  /// Server Invalid parameter value - TargetFrameNo outside of the allowed range 0..254 or does not exist on the RC
  /// Command "CalculateCartesianPosition"
  ERR_INVALID_PARAM_TARGET_FRAMENO_OUT_OF_RANGE := 16#8D72,

  /// Server Invalid parameter value - ToolNo outside of the allowed range 0..254 or does not exist on the RC
  /// Command "CalculateCartesianPosition"
  ERR_INVALID_PARAM_ERR_TOOLNO_INVALID := 16#8D73,

  /// Server Invalid parameter value - ParameterID does not exist on the RC
  /// Commands: "ReadSystemVariable", "WriteSystemVariable"
  ERR_INVALID_PARAM_PARAMETER_ID_INVALID := 16#8D74,

  /// Server Invalid parameter value - SubParameterID does not exist on the RC for the supplied ParameterID
  /// Commands: "ReadSystemVariable", "WriteSystemVariable"
  ERR_INVALID_PARAM_SUB_PARAMETER_ID_INVALID := 16#8D75,

  /// Server Invalid parameter value - SubParameterID must be 0 for a parameter without subparameters
  /// Commands: "ReadSystemVariable", "WriteSystemVariable"
  ERR_INVALID_PARAM_SUB_PARAMETER_MUST_BE_ZERO := 16#8D76,

  /// Server Invalid parameter value - SubParameterID must not be 0 for a parameter with subparameters
  /// Commands: "ReadSystemVariable", "WriteSystemVariable"
  ERR_INVALID_PARAM_SUB_PARAMETER_MUST_NOT_BE_ZERO := 16#8D77,

  /// Server Invalid parameter value - DataType outside of the allowed range 1..13
  /// Command "WriteSystemVariable"
  ERR_INVALID_PARAM_DATA_TYPE_OUT_OF_RANGE := 16#8D78,

  /// Server Invalid parameter value - DataType does not match the data type of the parameter
  /// Command "WriteSystemVariable"
  ERR_INVALID_PARAM_DATA_TYPE_MISMATCH := 16#8D79,

  /// Server Invalid parameter value - Data_0 contains invalid data for the target parameter
  /// Command "WriteSystemVariable"
  ERR_INVALID_PARAM_DATA_0_INVALID := 16#8D80,

  /// Server Invalid parameter value - Data_1 contains invalid data for the target parameter
  /// Command "WriteSystemVariable"
  ERR_INVALID_PARAM_DATA_1_INVALID := 16#8D81,

  /// Server Invalid parameter value - Data_2 contains invalid data for the target parameter
  /// Command "WriteSystemVariable"
  ERR_INVALID_PARAM_DATA_2_INVALID := 16#8D82,

  /// Server Invalid parameter value - Data_3 contains invalid data for the target parameter
  /// Command "WriteSystemVariable"
  ERR_INVALID_PARAM_DATA_3_INVALID := 16#8D83,

  /// Server Invalid parameter value - Data_4 contains invalid data for the target parameter
  /// Command "WriteSystemVariable"
  ERR_INVALID_PARAM_DATA_4_INVALID := 16#8D84,

  /// Server Invalid parameter value - Data_5 contains invalid data for the target parameter
  /// Command "WriteSystemVariable"
  ERR_INVALID_PARAM_DATA_5_INVALID := 16#8D85,

  /// Server Invalid parameter value - Data_6 contains invalid data for the target parameter
  /// Command "WriteSystemVariable"
  ERR_INVALID_PARAM_DATA_6_INVALID := 16#8D86,

  /// Server Invalid parameter value - Data_7 contains invalid data for the target parameter
  /// Command "WriteSystemVariable"
  ERR_INVALID_PARAM_DATA_7_INVALID := 16#8D87,

  /// Server Invalid parameter value - ReferenceFrame outside of the allowed range 0..254 or does not exist on the RC
  /// Command "CalculateFrame"
  ERR_INVALID_PARAM_REFERENCE_FRAME_OUT_OF_RANGE := 16#8D88,

  /// Server Optional parameter value not supported - DecelerationRate
  /// Commands using the parameter "DecelerationRate"
  ERR_OPTIONAL_PARAM_DECELERATION_RATE_NOT_SUPPORTED := 16#8E03,

  /// Server Optional parameter value not supported - JerkRate
  /// Commands using the parameter "JerkRate"
  ERR_OPTIONAL_PARAM_JERK_RATE_NOT_SUPPORTED := 16#8E04,

  /// Server Optional parameter value not supported - BlendingMode
  /// Commands using the parameter "BlendingMode"
  ERR_OPTIONAL_PARAM_BLENDING_MODE_NOT_SUPPORTED := 16#8E05,

  /// Server Optional parameter value not supported - Time
  /// Commands using the parameter "Time"
  ERR_OPTIONAL_PARAM_TIME_NOT_SUPPORTED := 16#8E06,

  /// Server Optional parameter value not supported - Position
  /// Commands using the parameter "Position"
  ERR_OPTIONAL_PARAM_POSITION_NOT_SUPPORTED := 16#8E07,

  /// Server Optional parameter value not supported - OriMode
  /// Commands using the parameter "OriMode"
  ERR_OPTIONAL_PARAM_ORI_MODE_NOT_SUPPORTED := 16#8E08,

  /// Server Optional parameter value not supported - ConfigMode
  /// Commands using the parameter "ConfigMode"
  ERR_OPTIONAL_PARAM_CONFIG_MODE_NOT_SUPPORTED := 16#8E09,

  /// Server Optional parameter value not supported - TurnMode
  /// Commands using the parameter "TurnMode"
  ERR_OPTIONAL_PARAM_TURN_MODE_NOT_SUPPORTED := 16#8E10,

  /// Server Optional parameter value not supported - TrajectoryMode
  /// Command "ReturnToPrimary"
  ERR_OPTIONAL_PARAM_TRAJECTORY_MODE_NOT_SUPPORTED := 16#8E11,

  /// Server Optional parameter value not supported - OperationMode
  /// Command "SetOperationMode"
  ERR_OPTIONAL_PARAM_OPERATION_MODE_NOT_SUPPORTED := 16#8E12,

  /// Server Optional parameter value not supported - IncrementalRotation
  /// Command "GroupJog"
  ERR_OPTIONAL_PARAM_INC_ROTATION_NOT_SUPPORTED := 16#8E13,

  /// Server Optional parameter value not supported - IncrementalTranslation
  /// Command "GroupJog"
  ERR_OPTIONAL_PARAM_INC_TRANSLATION_NOT_SUPPORTED := 16#8E14,

  /// Server Optional parameter value not supported - StepMode Exact Stop
  /// Command "EnableRobot"
  ERR_OPTIONAL_PARAM_STEP_MODE_EXACT_STOP_NOT_SUPPORTED := 16#8E16,

  /// Server Optional parameter value not supported - StepMode Blending
  /// Command "EnableRobot"
  ERR_OPTIONAL_PARAM_STEP_MODE_BLENDING_NOT_SUPPORTED := 16#8E17,

  /// Server Optional parameter value not supported - ModifiedConvention
  /// Command "ReadDHParameter"
  ERR_OPTIONAL_PARAM_MODIFIED_CONVENTION_NOT_SUPPORTED := 16#8E20,

  /// Server Optional parameter value not supported - WaitAtBlendingPoint
  /// Command "ExchangeConfig"
  ERR_OPTIONAL_PARAM_WAIT_AT_BLENDING_POINT_NOT_SUPPORTED := 16#8E21,

  /// Server Optional parameter not supported - Angle
  /// Commands: "MoveCircularAbsolute", "MoveCircularRelative", "MoveCircularCam"
  ERR_OPTIONAL_PARAM_ANGLE_NOT_SUPPORTED := 16#8E23,

  /// Server Optional parameter not supported - PathChoice
  /// Commands: "MoveCircularAbsolute", "MoveCircularRelative", "MoveCircularCam"
  ERR_OPTIONAL_PARAM_PATH_CHOICE_NOT_SUPPORTED := 16#8E24,

  /// Server Optional parameter not supported - Tolerance
  /// Commands: "MoveCircularAbsolute", "MoveCircularRelative", "MoveCircularCam"
  ERR_OPTIONAL_PARAM_TOLERANCE_NOT_SUPPORTED := 16#8E25,

  /// Server Optional parameter not supported - TransformationParameter_2
  /// Command "ShiftPosition"
  ERR_OPTIONAL_PARAM_TRANSFORMATION_PARAM2_NOT_SUPPORTED := 16#8E26,

  /// Server Optional parameter not supported - RotationAngle
  /// Command "ShiftPosition"
  ERR_OPTIONAL_PARAM_ROTATION_ANGLE_NOT_SUPPORTED := 16#8E27,

  /// Server Optional parameter value not supported - Mode
  /// Commands: "CalculateTool", "CalculateFrame"
  ERR_OPTIONAL_PARAM_VALUE_NOT_SUPPORTED := 16#8E28,

  /// Server Optional parameter not supported - ExternalTCP
  /// Commands: "CalculateTool", "CalculateFrame"
  ERR_OPTIONAL_PARAM_EXTERNAL_TCP_NOT_SUPPORTED := 16#8E29,

  /// Server Optional parameter not supported - RelativePosition
  /// Commands using the parameter "RelativePosition"
  ERR_OPTIONAL_PARAM_RELATIVE_POS_NOT_SUPPORTED := 16#8E30,

  /// Server Specified Emitter ID must not be 0
  /// Commands using the parameter "EmitterID"
  ERR_EMITTER_ID_MUST_NOT_BE_ZERO := 16#8F04,

  /// Server Invalid parameter value - Execution mode
  /// All Commands
  ERR_INVALID_PARAM_EXECUTION_MODE := 16#8F10,

  /// Server Command not implemented
  /// All Commands
  ERR_CMD_NOT_IMPLEMENTED := 16#8F11,

  /// Server Only one instance of this command is allowed
  /// Commands: "EnableRobot", "GroupJog", "ReturnToPrimary", "ExchangeConfig"
  ERR_CMD_ONLY_ONE_INSTANCE_ALLOWED := 16#8F12,

  /// Server Command requires an active interrupt or idle state to be executed
  /// Commands: "GroupJog", "ReturnToPrimary"
  ERR_CMD_REQUIRES_INTERRUPT_OR_IDLE_STATE := 16#8F13,

  /// Server Command cannot be executed during active interrupt
  /// Command "ReturnToPrimary"
  ERR_CMD_NOT_ALLOWED_DURING_ACTIVE_INTERRUPT := 16#8F14,

  /// Server Secondary sequence is blocked by command (e.g. GroupJog, ReturnToPrimary). No other commands may be buffered in secondary sequence
  /// All commands processed in secondary sequence
  ERR_SECONDARY_SEQUENCE_BLOCKED_BY_CMD := 16#8F15,

  /// Server The secondary sequence is not active. Commands may only be buffered in this sequence if it is active
  /// Commands using the parameter "SequenceFlag"
  ERR_SECONDARY_SEQUENCE_NOT_ACTIVE := 16#8F16,

  /// Server Secondary sequence is not empty. The command requires the secondary sequence to be empty
  /// Commands: "GroupJog", "ReturnToPrimary"
  ERR_SECONDARY_SEQUENCE_NOT_EMPTY := 16#8F17,

  /// Server Transaction not possible in the state machine
  /// All commands
  ERR_TRANSACTION_NOT_POSSIBLE_IN_STATE_MACHINE := 16#8F18,

  /// Server Cannot execute command because current operation mode is local.
  /// Commands that are not available in local modes
  ERR_CMD_NOT_POSSIBLE_BY_OP_MODE_LOCAL := 16#8F19,

  /// Server Command type out of range
  /// All commands
  ERR_CMD_TYPE_OUT_OF_RANGE := 16#8F20,

  /// Server Execution of this CMD is not possible while CallSubprogram is in progress in the sequence
  /// Commands: "SetSequence", "GroupJog"
  ERR_CMD_NOT_POSSIBLE_DURING_CALL_SUB_PROGRAM := 16#8F21,

  /// Server Operation not possible. See MessageLog for further information
  /// All commands
  ERR_OPERATION_NOT_POSSIBLE_SEE_LOG := 16#8F36,

  /// Server An RC internal error occurred during execution of this command. Check the message log for additional information
  /// All commands
  ERR_INTERNAL_ERROR_DURING_CMD := 16#8FFF,
  
  /// 7.2 Table "B" – RI ErrorIDs
  /// RI errors can occur on the PLC as well as on the RC. In the event of an RI error on the PLC, the
  /// corresponding ErrorID is written to the PLC message buffer independent of the function call
  /// "ReadMessages". In the event of an RI error on the RC, the ErrorID is transmitted via the function
  /// block "ReadMessages" and is also stored in PLC message buffer.
  /// In the PLC message buffer, they are dynamically arranged by the client to be displayed as follows:
  /// <Origin> <MessageType> <Description>
  /// More information about the general message handling mechanism can be found in 5.5.11
  /// Diagnostics.
  /// The following table gives an overview over the existing "ErrorIDs" reported via RI errors and the
  /// corresponding description.

  /// ------------------------------------------------------
  /// Client ErrorIDs
  /// ------------------------------------------------------

  /// Client Wrong Telegram State (Two Sequences not in both directions active)
  ERR_WRONG_TELEGRAM_STATE  := 16#8001,

  /// Client Acyclic area client to server too small
  ERR_ACYCLIC_AREA_TO_SMALL_PLC_TO_ROB  := 16#8002,

  /// Client Acyclic area server to client too small
  ERR_ACYCLIC_AREA_TO_SMALL_ROB_TO_PLC := 16#8003,

  /// Client Lifesign timeout
  ERR_LIFESIGN_TIMEOUT_0x8005 := 16#8004,

  /// Client Telegram sequence timeout
  ERR_TELEGRAM_SEQ_TIMEOUT_0x8005 := 16#8005,

  /// Client Assigned AxesGroup not valid
  ERR_AXESGROUP_INVALID := 16#8007,

  /// Client Assigned periphery not valid
  ERR_PERIPHERY_INVALID := 16#8008,

  /// Client Invalid state of the robot (more than 1 CMD active)
  ERR_INVALID_ROBOT_STATE := 16#8009,

  /// Client Telegram Number changed after initialization. Reinitialize by disabling and enabling the RobotTask.
  ERR_TELEGRAM_NUMBER_CHANGED_AFTER_INIT  := 16#8013,
    
  /// Client Telegram control does not match the telegram state
  ERR_TELEGRAM_CONTROL_MISMATCH_TELEGRAM_STATE_0x80A1 := 16#80A1,

  /// Client Initialization lost for unknown reason. See message log after reinitializing
  ERR_INIT_LOST_UNKNOWN_0x80A2  := 16#80A2,

  /// Client Telegram length does not match the length provided in the communication interface, or the communication interface is too small.
  ERR_TELEGRAM_LENGTH_MISMATCH_0x80A3  := 16#80A3,

  /// Client Incompatible major SRCI version
  ERR_SRCI_MAJOR_VERSION_INCOMPATIBLE_0x80A4  := 16#80A4,

  /// Client Lifesign timeout
  ERR_LIFESIGN_TIMEOUT_0x80A5 := 16#80A5,

  /// Client The selected optional cyclic data does not fit in the given telegram size
  ERR_CYCLIC_DATA_TOO_LARGE_0x80A6  := 16#80A6,

  /// Client The robot interface was reset after being initialized
  ERR_INTERFACE_WAS_RESET_AFTER_INIT_0x80A7  := 16#80A7,

  /// Client Telegram sequence timeout
  ERR_TELEGRAM_SEQ_TIMEOUT_0x80A8_0x80A8  := 16#80A8,

  /// Client The telegram number changed after initialization
  ERR_TELEGRAM_NO_CHANGED_AFTER_INIT_0x80A9 := 16#80A9,

  /// Client Error: Invalid AxesGroupID
  ERR_AXESGROUP_ID_INVALID_0x80AA  := 16#80AA,

  /// Client Telegram number is invalid. E.g. TwoSequences is only activated in one direction
  ERR_TELEGRAM_NUMBER_INVALID_0x80AB  := 16#80AB,

  /// Client Telegram Number is not supported
  ERR_TELEGRAM_NUMBER_NOT_SUPPORTED_0x80AC := 16#80AC,

  /// Server The ACR is full. RA is disabled
  ERR_ACR_REGISER_IS_FULL  := 16#8A01,

  /// Server The execution of a mandatory command has been stopped. Exchange config must run for the system to run
  ERR_MANDATORY_CMD_STOPPED  := 16#8A02,

  /// Server Inconsistent data received. Make sure the complete telegram data is sent to RC in one frame.
  ERR_INCONSISTENT_DATA_RECEIVED  := 16#8A03,

  /// Client Connection to the communication partner was lost
  ERR_CONNECTION_LOST  := 16#8AAD,

  /// Client Fatal Error occurred. Reinitialization of Robot_Task is required
  ERR_FATAL_ERROR_REINIT_REQUIRED  := 16#9001,

  /// ------------------------------------------------------
  /// SERVER ErrorIDs
  /// ------------------------------------------------------
  
  /// Server Internal error
  ERR_INTERNAL_ERROR  := 16#9A01,

  /// Server Internal error in deserialize
  ERR_DESERIALIZE_ERROR  := 16#9A02,

  /// Server CMD ID out of range 1.ACR_Length
  ERR_CMD_ID_OUT_OF_RANGE  := 16#9A03,

  /// Server Invalid fragment length
  ERR_FRAGMENT_LENGTH_INVALID := 16#9A04,

  /// Server Command priority or type changed during runtime
  ERR_CMD_PRIORITY_CHANGED := 16#9A05,

  /// Server Tried to reset a non-empty ACR entry
  ERR_TRIED_TO_RESET_NONEMPTY_ACR_REGISTER := 16#9A06,

  /// Server Error: Invalid Sequence payload length (e.g., sequence payload length is specified 999 even if telegram length is only 100.)
  ERR_SEQUENCE_PAYLOAD_INVALID_LENGTH := 16#9A07,

  /// Server Invalid ActionByte
  ERR_ACTION_BYTE_INVALID := 16#9A08,

  /// Server Invalid Command payload length
  ERR_CMD_PAYLOAD_LENGTH_INVALID := 16#9A09,

  /// Server Error: Invalid Command payload pointer (e.g., Out of bounds)
  ERR_CMD_PAYLOAD_POINTER_INVALID := 16#9A10,

  /// Server Illegal Execution Mode change
  ERR_EXEC_MODE_CHANGE_ILLEGAL := 16#9A14

)WORD;
END_TYPE

// Library/Enumerations/Events/RobotLibraryInfoIdEnum
{attribute 'qualified_only'}
TYPE RobotLibraryInfoIdEnum :
(
  NO_INFO := 0,
  
  ////7.5 Table "E" – Command InfoIDs
  /// If an info event related to the execution of a function block occurs, the function block returns an
  /// InfoID to specify the event. The info events are stored in the PLC message buffer and are displayed
  /// on the function block outputs.
  /// In the PLC message buffer, they are dynamically arranged by the client to be displayed as follows:
  /// <Origin> <MessageType> <Command name> <Description>
  /// More information about the general message handling mechanism can be found in 5.5.11
  /// Diagnostics.
  /// The following table gives an overview over the existing InfoIDs reported by commands and the
  /// corresponding description.

  /// Server Collision detected
  /// Motion commands
  INFO_COLLISION_DETECTED := 16#6C01,

  /// Server Error occurred during motion. Check the message buffer for more information
  /// Motion commands
  INFO_MOTION_ERROR := 16#6C02,

  /// Server Target position not reachable
  /// Motion commands
  INFO_TARGET_POS_UNREACHABLE := 16#6C03,

  /// Server Software limits reached
  /// Motion commands
  INFO_SW_LIMITS_REACHED := 16#6C04,

  /// Server Abortion of this command was requested by a GroupStop
  /// All sequence related commands
  INFO_ABORT_BY_GROUP_STOP := 16#6C05,

  /// Server Abortion of this command was requested by another motion command
  /// All sequence related commands
  INFO_ABORT_BY_MOTION_CMD := 16#6C06,

  /// Server Reading the currently used software limits. Updated software limits are active after restart.
  /// Command "ReadRobotSWLimits"
  INFO_READ_SW_LIMITS := 16#6C07,

  /// Server No SubProgram was stopped because none was active
  /// Command "StopSubprogram"
  INFO_NO_ACTIVE_SUBPROGRAM := 16#6C09,

  /// Server A program for the supplied JobID is not running or does not exist.
  /// Command "StopSubprogram"
  INFO_JOBID_NOT_RUNNING := 16#6C11,

  /// Server A program for the supplied InstanceID is not running or does not exist.
  /// Command "StopSubprogram"
  INFO_INSTANCEID_NOT_RUNNING := 16#6C12,

  /// Server The robot is waiting at the blending zone.
  /// Motion commands
  INFO_WAITING_AT_BLEND_ZONE := 16#6C13,

  /// Server Jog motion was interrupted by GroupStop
  /// Command "GroupJog"
  INFO_JOG_INTERRUPTED_BY_GROUP_STOP := 16#6C14,

  /// Server Jog motion was interrupted by RA sequence state INTERRUPTED
  /// Command "GroupJog"
  INFO_JOG_INTERRUPTED_BY_RA_STATE := 16#6C15,

  /// Server Manual start is ignored when the sequence is empty
  /// Command "EnableRobot"
  INFO_MANUAL_START_IGNORED_DURING_EMPTY_SEQ := 16#6C19,

  /// Server Invalid parameter value - A value was given for index 0. Index 0 is not writeable. Remove the value or change the index.
  /// Commands: "WriteIntegers", "WriteReals", "WriteAnalogOutputs", "ReadDigitalInputs", "ReadDigitalOutputs", "ReadIntegers", "ReadReals"
  INFO_PARAM_INDEX_ZERO_NOT_WRITEABLE := 16#6D51,

  /// Server Invalid parameter value OutputBitmask - No bitmask was given for a non zero index. Set the index to zero, or set a valid bitmask.
  /// Command "WriteDigitalOutputs"
  INFO_PARAM_OUTPUT_BITMASK_INVALID_FOR_NON_ZERO_INDEX := 16#6D52,

  /// Server Invalid parameter value OutputBitmask - A bitmask was given for a zero index. Set the bitmask to zero, or set a non zero index.
  /// Command "WriteDigitalOutputs"
  INFO_PARAM_OUTPUT_BITMASK_INVALID_FOR_ZERO_INDEX := 16#6D53,

  /// Server Command interrupted due to RA sequence state INTERRUPTED
  /// All sequence related commands
  INFO_CMD_INTERRUPTED_BY_RA_STATE  := 16#6F01,

  /// Server Command interrupted due to RA power state NOT_ENABLED
  /// All sequence related commands
  INFO_CMD_INTERRUPTED_BY_RA_NOT_ENABLED  := 16#6F02,

  /// Server Command interrupted due to RA sequence state INTERRUPTED while single step mode is active
  /// All sequence related commands
  INFO_CMD_INTERRUPTED_BY_RA_SEQ_STATE_DURING_STEP_MODE  := 16#6F03,

  /// Server Internal code used to reset warnings
  /// All commands
  INFO_RESET_WARNINGS_BY_INTERNAL_CODE  := 16#FF,


  /// 7.6 Table "F" – RI InfoIDs
  /// RI info events can occur on the PLC as well as on the RC. In the event of an RI info on the PLC,
  /// the corresponding InfoID is written to the PLC message buffer independent of the function call
  /// "ReadMessages". In the event of an RI info on the RC, the InfoID is transmitted via the function
  /// block "ReadMessages" and is also stored in PLC message buffer.
  /// In the PLC message buffer, they are dynamically arranged by the client to be displayed as follows:
  /// <Origin> <MessageType> <Description>
  /// More information about the general message handling mechanism can be found in 5.5.11
  /// Diagnostics.
  /// The following table gives an overview over the existing InfoIDs reported via RI info events and the
  /// corresponding description.  

  /// Client Lifesign smaller than lower limit. It has been increased to 10ms.
  INFO_LIFESIGN_TIMEOUT_TO_SMALL_AND_SET_TO_10MS  := 16#6001,

  /// Client ReceiveExtendedCartesianPosition cannot be used without ReceiveCartesianPos. RecCarPos is automatically activated.
  INFO_RECV_EXT_CART_POS_NOT_USABLE_WITH_RECV_CART_POS := 16#6002,

  /// Client ReceiveExtendedJointPosition cannot be used without ReceiveJointPosition. RecJointPos is automatically activated.
  INFO_RECV_EXT_JOINT_POS_NOT_USABLE_WITH_RECV_JOINT_POS := 16#6003,

  /// Client Synchronization of tool data is disabled, and the data is different on the RC. Tool = "NUMBER" (Please Enter a valid SyncMode)
  INFO_SYNC_TOOL_DATA_DISABLED  := 16#6014,

  /// Client Change the Syncmode to Negative only works on Startup with PLC (TOOL)
  INFO_CHANGE_TOOL_SYNC_MODE_TO_NEGATIVE_ONLY_AT_PLC_START_ALLOWED := 16#6015,

  /// Client Synchronization of frame data is disabled, and the data is different on the RC. Frame = "NUMBER" (Please Enter a valid SyncMode)
  INFO_SYNC_FRAME_DATA_DISABLED := 16#6020,

  /// Client Change the Syncmode to Negative only works on Startup with PLC (FRAME)
  INFO_CHANGE_FRAME_SYNC_MODE_TO_NEGATIVE_ONLY_AT_PLC_START_ALLOWED := 16#6021,

  /// Client Synchronization of load data is disabled, and the data is different on the RC. Load = "NUMBER" (Please Enter a valid SyncMode)
  INFO_SYNC_LOAD_DATA_DISABLED := 16#6026,

  /// Client Change the Syncmode to Negative only works on Startup with PLC (LOAD)
  INFO_CHANGE_LOAD_SYNC_MODE_TO_NEGATIVE_ONLY_AT_PLC_START_ALLOWED := 16#6027,

  /// Client Synchronization of work area data is disabled, and the data is different on the RC. WorkArea = "NUMBER" (Please Enter a valid SyncMode)
  INFO_SYNC_WORK_AREA_DISABLED := 16#6032,

  /// Client Change the Syncmode to Negative only works on Startup with PLC (WORKAREA)
  INFO_CHANGE_WORK_AREA_SYNC_MODE_TO_NEGATIVE_ONLY_AT_PLC_START_ALLOWED := 16#6033,

  /// Client Synchronization of Software Limits data is disabled, and the data is different on the RC.
  INFO_SYNC_SWLIMIT_DISABLED := 16#6036,

  /// Client Change the Syncmode to Negative only works on Startup with PLC (SW LIMITS)
  INFO_CHANGE_SWLIMITS_SYNC_MODE_TO_NEGATIVE_ONLY_AT_PLC_START_ALLOWED := 16#6037,

  /// Client Synchronization of default dynamics data is disabled, and the data is different on the RC.
  INFO_SYNC_DEFAULT_DYNAMICS_DISABLED := 16#6040,

  /// Client Change the Syncmode to Negative only works on Startup with PLC (DEFAULT DYNAMICS)
  INFO_CHANGE_DEFAULT_DYNAMIVS_SYNC_MODE_TO_NEGATIVE_ONLY_AT_PLC_START_ALLOWED := 16#6041,

  /// Client Synchronization of reference dynamics data is disabled, and the data is different on the RC.
  INFO_SYNC_REFERENCE_DYNAMICS_DISABLED := 16#6044,

  /// Client Change the Syncmode to Negative only works on Startup with PLC (REFERENCE DYNAMICS)
  INFO_CHANGE_REFERENCE_DYNAMIVS_SYNC_MODE_TO_NEGATIVE_ONLY_AT_PLC_START_ALLOWED := 16#6045,

  /// Server RA disabled due to operation mode change
  INFO_RA_DISABLED_BY_OPMODE_CHANGE  := 16#6A01,

  /// Server Operation mode changed
  INFO_OPERATION_MODE_CHANGED  := 16#6A02,

  /// Server The server state has been reset on client request. Client restart may be a cause.
  INFO_SERVER_STATE_RESET_BY_CLIENT_REQUEST  := 16#6A03,

  /// Server The actual override has been decreased to not exceed a movement's monitoring velocity.
  INFO_OVERRIDE_DECREASED_TO_PREVENT_EXEEDING_MONITORING_VELOCITY  := 16#6A07,

  /// Server Excessive logging may degrade system performance.
  INFO_EXCESSIVE_LOGGING  := 16#6A13,

  /// Server The first motion is executed with reduced velocity.
  INFO_FIRST_MOTION_REDUCED_VELOCITY  := 16#6C08
)WORD;
END_TYPE

// Library/Enumerations/Events/RobotLibraryWarningIdEnum
{attribute 'qualified_only'}
TYPE RobotLibraryWarningIdEnum :
(
  NO_WARNING := 0,
 
  /// 7.3 Table "C" – Command WarningIDs
  /// If a warning related to the execution of a function block occurs, the function block returns a
  /// WarningID to specify the warning. The warnings are stored in the PLC message buffer and are
  /// displayed on the function block outputs.
  /// In the PLC message buffer, they are dynamically arranged by the client to be displayed as follows:
  /// <Origin> <MessageType> <Command name> <Description>
  /// More information about the general message handling mechanism can be found in 5.5.11
  /// Diagnostics.
  /// The following table gives an overview over the existing WarningIDs reported by commands and
  /// the corresponding description.

  /// Client HighPriority Input is ignored when a sequential ProcessingMode is selected
  /// Commands: "WriteDigitalOutputs", "WriteIntegers", "WriteReals", "WriteAnalogOutputs"
  WARN_HIGHPRIORITY_IGNORED_SEQ_MODE  := 16#7301,

  /// Client Optional Cyclic data was disabled by the user but is still enabled until reinitialization of RobotTask
  /// Command: "ReadActualPositionCyclic"
  WARN_CYCLIC_DATA_DISABLED_STILL_ACTIVE  := 16#7303,

  /// Client Number of free entries in the ACR is running out
  /// All commands
  WARN_ACR_FREE_ENTRIES_LOW  := 16#7605,

  /// Server The Frame is currently used in the sequence
  /// Command: "WriteFrameData"
  WARN_FRAME_USED_IN_SEQUENCE  := 16#7C03,

  /// Server The Tool is currently used in the sequence
  /// Command: "WriteToolData"
  WARN_TOOL_USED_IN_SEQUENCE  := 16#7C04,

  /// Server The Load is currently used in the sequence
  /// Command: "WriteLoadData"
  WARN_LOAD_USED_IN_SEQUENCE  := 16#7C06,

  /// Server The monitoring does not apply to motion CMDs which are already buffered.
  /// Command: "SetTriggerMotion"
  WARN_MONITORING_DOES_NOT_APPLY_TO_BUFFERED_CMDS  := 16#7C14,

  /// 7.4 Table "D" – RI WarningIDs
  /// RI warnings can occur on the PLC as well as on the RC. In the event of an RI warning on the PLC,
  /// the corresponding WarningID is written to the PLC message buffer independent of the function call
  /// "ReadMessages". In the event of an RI warning on the RC, the WarningID is transmitted via the
  /// function block "ReadMessages" and is also stored in PLC message buffer.
  /// In the PLC message buffer, they are dynamically arranged by the client to be displayed as follows:
  /// <Origin> <MessageType> <Description>
  /// More information about the general message handling mechanism can be found in 5.5.11
  /// Diagnostics.
  /// The following table gives an overview over the existing WarningIDs reported via RI warnings and
  /// the corresponding description.

  /// Client Acyclic range client to server very small
  WARN_ACYCLIC_RANGE_PLC_TO_ROB_VERY_SMALL  := 16#7001,

  /// Client Acyclic range server to client very small
  WARN_ACYCLIC_RANGE_ROB_TO_PLC_VERY_SMALL := 16#7002,

  /// Client Telegram number was changed during operation
  WARN_TELEGRAM_NO_CHANGED_DURING_OPERATION  := 16#7003,

  /// Client Save Tool locally failed. Index not available in user data.
  WARN_SAVE_TOOL_FAILED := 16#7005,

  /// Client Save Frame locally failed. Index not available in user data.
  WARN_SAVE_FRAME_FAILED  := 16#7006,

  /// Client Save Load locally failed. Index not available in user data.
  WARN_SAVE_LOAD_FAILED  := 16#7007,

  /// Client Save WorkArea locally failed. Index not available in user data.
  WARN_SAVE_WORKAREA_FAILED  := 16#7008,

  /// Client Array of tool data supplied to RobotTask does not start at 0.
  WARN_TOOL_DATA_ARRAY_NOT_START_AT_ZERO  := 16#7009,

  /// Client Array of tool data supplied to RobotTask must be longer than the number of tools on the RC.
  WARN_TOOL_DATA_ARRAY_TOO_SHORT := 16#7010,

  /// Client Tool data sync mode is invalid.
  WARN_TOOL_DATA_SYNC_MODE_INVALID  := 16#7011,

  /// Client Error Sync with Tool "NUMBER" (Please Enter a valid SyncMode)
  WARN_TOOL_NUMBER_SYNC_ERROR  := 16#7012,

  /// Client Error Sync Data changed in both Sides with Tool "NUMBER" (Please Enter a valid SyncMode)
  WARN_TOOL_SYNC_BOTH_SIDES_CHANGED  := 16#7013,

  /// Client Array of frame data supplied to RobotTask does not start at 0.
  WARN_FRAME_DATA_ARRAY_NOT_START_AT_ZERO := 16#7015,

  /// Client Array of frame data supplied to RobotTask must be longer than the number of frames on the RC.
  WARN_FRAME_DATA_ARRAY_TOO_SHORT := 16#7016,

  /// Client Frame data sync mode is invalid.
  WARN_FRAME_DATA_SYNC_MODE_INVALID := 16#7017,

  /// Client Error Sync with Frame "NUMBER" (Please Enter a valid SyncMode)
  WARN_FRAME_NUMBER_SYNC_ERROR := 16#7018,

  /// Client Error Sync Data changed in both Sides with Frame "NUMBER" (Please Enter a valid SyncMode)
  WARN_FRAME_SYNC_BOTH_SIDES_CHANGED := 16#7019,

  /// Client Array of load data supplied to RobotTask does not start at 0.
  WARN_LOAD_DATA_ARRAY_NOT_START_AT_ZERO := 16#7021,

  /// Client Array of load data supplied to RobotTask must be longer than the number of tools on the RC.
  WARN_LOAD_DATA_ARRAY_TOO_SHORT := 16#7022,

  /// Client Load data sync mode is invalid.
  WARN_LOAD_DATA_SYNC_MODE_INVALID := 16#7023,

  /// Client Error Sync with Load "NUMBER" (Please Enter a valid SyncMode)
  WARN_LOAD_NUMBER_SYNC_ERROR := 16#7024,

  /// Client Error Sync Data changed in both Sides with Load "NUMBER" (Please Enter a valid SyncMode)
  WARN_LOAD_SYNC_BOTH_SIDES_CHANGED := 16#7025,

  /// Client Array of workarea data supplied to RobotTask does not start at 0.
  WARN_WORK_AREA_ARRAY_NOT_START_AT_ZERO := 16#7027,

  /// Client Array of workarea data supplied to RobotTask must be longer than the number of tools on the RC.
  WARN_WORK_AREA_ARRAY_TOO_SHORT := 16#7028,

  /// Client Workarea data sync mode is invalid.
  WARN_WORK_AREA_SYNC_MODE_INVALID := 16#7029,

  /// Client Error Sync with WorkArea "NUMBER" (Please Enter a valid SyncMode)
  WARN_WORK_AREA_NUMBER_SYNC_ERROR:= 16#7030,

  /// Client Error Sync Data changed in both Sides with WorkArea "NUMBER" (Please Enter a valid SyncMode)
  WARN_WORK_AREA_SYNC_BOTH_SIDES_CHANGED := 16#7031,

  /// Client Software limits data sync mode is invalid.
  WARN_SW_LIMITS_SYNC_MODE_INVALID := 16#7033,

  /// Client Error Sync with Software Limits (Please Enter a valid SyncMode)
  WARN_SW_LIMITS_SYNC_ERROR := 16#7034,

  /// Client Error Sync Data changed in both Sides with Software Limits (Please Enter a valid SyncMode)
  WARN_SW_LIMITS_SYNC_BOTH_SIDES_CHANGED := 16#7035,

  /// Client Default dynamics data sync mode is invalid.
  WARN_DEFAULT_DYNAMICS_SYNC_MODE_INVALID := 16#7037,

  /// Client Error Sync with Default Dynamics (Please Enter a valid SyncMode)
  WARN_DEFAULT_DYNAMICS_SYNC_ERROR := 16#7038,

  /// Client Error Sync Data changed in both Sides with Default Dynamics (Please Enter a valid SyncMode)
  WARN_DEFAULT_DYNAMICS_SYNC_BOTH_SIDES_CHANGED := 16#7039,

  /// Client Reference dynamics data sync mode is invalid.
  WARN_REFERENCE_DYNAMICS_SYNC_MODE_INVALID := 16#7041,

  /// Client Error Sync with Reference Dynamics (Please Enter a valid SyncMode)
  WARN_REFERENCE_DYNAMICS_SYNC_ERROR:= 16#7042,

  /// Client Error Sync Data changed in both Sides with Reference Dynamics (Please Enter a valid SyncMode)
  WARN_REFERENCE_DYNAMICS_SYNC_BOTH_SIDES_CHANGED := 16#7043,

  /// Client Synchronization of tool is not possible due to error in the read or write tool cmd. See dedicated message log entry for more information.
  WARN_TOOL_SYNC_FAILED_BY_ERROR_OF_READ_OR_WRITE_CMD  := 16#7044,

  /// Client Synchronization of frame is not possible due to error in the read or write frame cmd. See dedicated message log entry for more information.
  WARN_FRAME_SYNC_FAILED_BY_ERROR_OF_READ_OR_WRITE_CMD := 16#7045,

  /// Client Synchronization of load is not possible due to error in the read or write load cmd. See dedicated message log entry for more information.
  WARN_LOAD_SYNC_FAILED_BY_ERROR_OF_READ_OR_WRITE_CMD := 16#7046,

  /// Client Synchronization of swLimits is not possible due to error in the read or write swLimits cmd. See dedicated message log entry for more information.
  WARN_SW_LIMITS_SYNC_FAILED_BY_ERROR_OF_READ_OR_WRITE_CMD := 16#7047,

  /// Client Synchronization of referenceDynamics is not possible due to error in the read or write referenceDynamics cmd. See dedicated message log entry for more information.
  WARN_REFERENCE_DYNAMICS_SYNC_FAILED_BY_ERROR_OF_READ_OR_WRITE_CMD := 16#7048,

  /// Client Synchronization of defaultDynamics is not possible due to error in the read or write defaultDynamics cmd. See dedicated message log entry for more information.
  WARN_DEFAULT_DYNAMICS_SYNC_FAILED_BY_ERROR_OF_READ_OR_WRITE_CMD := 16#7049,

  /// Client Using the legacy SRCI version encoding. It will not be compatible with the newest RC interpreter versions.
  WARN_LEGACY_SRCI_ENCODING  := 16#7050,

  /// Server The ACR is almost full. Filling it completely disables the robot. Make sure to limit the number of commands in the system.
  WARN_ACR_ALMOST_FULL  := 16#7A01
)WORD;
END_TYPE

// Library/Enumerations/Flag/SequenceFlag
{attribute 'qualified_only'}
// ------------------------------------------------------------------------- 
//  SRCI Robot Library                                                
// ------------------------------------------------------------------------- 
//                                                                           
//  Object:      SequenceFlag                                       
//  Author:      Thorsten Brach                                                
//  Date:        2024-06-01
//
//  Description:                                              
//   
//                                                                           
//  Copyright: 
//    (C) 2024 Thorsten Brach. All rights reserved                                                                                                                                            
//             Licensed under the LGPL-3.0 license.
//                                                                           
//  Disclaimer:                                                                           
//    This project is provided without any guarantee and can be used for   
//    private and commercial purposes. Any use is at the user’s 
//    own risk and responsibility.
//
// -------------------------------------------------------------------------
TYPE SequenceFlag :
(
  /// • Refers to ProcessingModes 2 to 5 and 9 (2 = Parallel, 3 = Continuous, 4 = not available, 5 = Trigger Multiple, 9 = Deactivate )
  /// • Command is not handled by any sequence
  /// • For more information on ProcessingModes refer to chapter 5.6.4.5
  NO_SEQUENCE := 0,
  /// • Command will be handled by primary sequence
  PRIMARY_SEQUENCE := 1,
  /// • Command will be handled by secondary sequence
  SECONDARY_SEQUENCE := 2
)USINT;
END_TYPE

// Library/Enumerations/Level/LogLevel
{attribute 'qualified_only'}
// ------------------------------------------------------------------------- 
//  SRCI Robot Library                                                
// ------------------------------------------------------------------------- 
//                                                                           
//  Object:      LogLevel                                       
//  Author:      Thorsten Brach                                                
//  Date:        2024-06-01
//
//  Description:                                              
//   
//                                                                           
//  Copyright: 
//    (C) 2024 Thorsten Brach. All rights reserved                                                                                                                                            
//             Licensed under the LGPL-3.0 license.
//                                                                           
//  Disclaimer:                                                                           
//    This project is provided without any guarantee and can be used for   
//    private and commercial purposes. Any use is at the user’s 
//    own risk and responsibility.
//
// -------------------------------------------------------------------------
TYPE LogLevel : Severity; END_TYPE

// Library/Enumerations/Level/LogLevelEnum
TYPE LogLevelEnum : LogLevel; END_TYPE

// Library/Enumerations/Level/MessageLevel
{attribute 'qualified_only'}
// ------------------------------------------------------------------------- 
//  SRCI Robot Library                                                
// ------------------------------------------------------------------------- 
//                                                                           
//  Object:      MessageLevel                                       
//  Author:      Thorsten Brach                                                
//  Date:        2024-06-01
//
//  Description:                                              
//   
//                                                                           
//  Copyright: 
//    (C) 2024 Thorsten Brach. All rights reserved                                                                                                                                            
//             Licensed under the LGPL-3.0 license.
//                                                                           
//  Disclaimer:                                                                           
//    This project is provided without any guarantee and can be used for   
//    private and commercial purposes. Any use is at the user’s 
//    own risk and responsibility.
//
// -------------------------------------------------------------------------
TYPE MessageLevel :
(
  /// Debugging messages, Informative messages, Warning messages, Error messages, Fatal error messages
  DEBUG := 4,
  /// Informative messages, Warning messages, Error messages, Fatal error messages 
  INFO := 5, 
  /// Warning messages, Error messages, Fatal error messages
  WARNING := 20,
  /// Error messages, Fatal error messages 
  ERROR := 28 
)USINT;
END_TYPE

// Library/Enumerations/Level/PriorityLevel
{attribute 'qualified_only'}
// ------------------------------------------------------------------------- 
//  SRCI Robot Library                                                
// ------------------------------------------------------------------------- 
//                                                                           
//  Object:      PriorityLevel                                       
//  Author:      Thorsten Brach                                                
//  Date:        2024-06-01
//
//  Description:                                              
//   
//                                                                           
//  Copyright: 
//    (C) 2024 Thorsten Brach. All rights reserved                                                                                                                                            
//             Licensed under the LGPL-3.0 license.
//                                                                           
//  Disclaimer:                                                                           
//    This project is provided without any guarantee and can be used for   
//    private and commercial purposes. Any use is at the user’s 
//    own risk and responsibility.
//
// -------------------------------------------------------------------------
TYPE PriorityLevel :
(
  /// priority level is very high 
  VERY_HIGH := 1,
  /// priority level is high 
  HIGH := 2,
  /// priority level is normal 
  NORMAL := 3,
  /// priority level is low 
  LOW := 4  
)BYTE;
END_TYPE

// Library/Enumerations/Miscellaneous/CircPlane
{attribute 'qualified_only'}
{attribute 'strict'}
// ------------------------------------------------------------------------- 
//  SRCI Robot Library                                                
// ------------------------------------------------------------------------- 
//                                                                           
//  Object:      CircPlane                                       
//  Author:      Thorsten Brach                                                
//  Date:        2024-06-01
//
//  Description:                                              
//   
//                                                                           
//  Copyright: 
//    (C) 2024 Thorsten Brach. All rights reserved                                                                                                                                            
//             Licensed under the LGPL-3.0 license.
//                                                                           
//  Disclaimer:                                                                           
//    This project is provided without any guarantee and can be used for   
//    private and commercial purposes. Any use is at the user’s 
//    own risk and responsibility.
//
// -------------------------------------------------------------------------
TYPE CircPlane :
(
  /// x-z-plane
  XZ_PLANE := 0,
  /// y-z-plane
  YZ_PLANE := 1,
  /// x-y-plane
  XY_PLANE := 2
)SINT;
END_TYPE

// Library/Enumerations/Miscellaneous/ControlHalfByte
{attribute 'qualified_only'}
// ------------------------------------------------------------------------- 
//  SRCI Robot Library                                                
// ------------------------------------------------------------------------- 
//                                                                           
//  Object:      ControlHalfByte                                       
//  Author:      Thorsten Brach                                                
//  Date:        2024-06-01
//
//  Description:                                              
//   
//                                                                           
//  Copyright: 
//    (C) 2024 Thorsten Brach. All rights reserved                                                                                                                                            
//             Licensed under the LGPL-3.0 license.
//                                                                           
//  Disclaimer:                                                                           
//    This project is provided without any guarantee and can be used for   
//    private and commercial purposes. Any use is at the user’s 
//    own risk and responsibility.
//
// -------------------------------------------------------------------------
TYPE ControlHalfByte :
(
  /// Default value, no control active
  NONE := 0,
  /// Initialization is requested by the client
  INITIALIZE := 1,
  /// Resume of operation is requested by the client
  RESUME := 2,
  /// Resetting of the RC is requested by the client. The RC must stop the motion, and clear all state.
  RESET := 3,
  /// Acknowledgement of a telegram state error
  ACK_ERROR := 4,
  /// Signaling that a client error occurred. The Server must respond by setting its RI state to NOT_INITIALIZED
  CLIENT_ERROR := 5
)BYTE;
END_TYPE

// Library/Enumerations/Miscellaneous/ErrorReaction
{attribute 'qualified_only'}
// ------------------------------------------------------------------------- 
//  SRCI Robot Library                                                
// ------------------------------------------------------------------------- 
//                                                                           
//  Object:      ErrorReaction                                       
//  Author:      Thorsten Brach                                                
//  Date:        2024-06-01
//
//  Description:                                              
//   
//                                                                           
//  Copyright: 
//    (C) 2024 Thorsten Brach. All rights reserved                                                                                                                                            
//             Licensed under the LGPL-3.0 license.
//                                                                           
//  Disclaimer:                                                                           
//    This project is provided without any guarantee and can be used for   
//    private and commercial purposes. Any use is at the user’s 
//    own risk and responsibility.
//
// -------------------------------------------------------------------------
TYPE ErrorReaction :
(
  /// Abort and move Abort active move command and delete commands buffered in sequence Move robot by specified ErrorVector
  ABORT_AND_MOVE := 0,
  /// 1: Abort
  /// Abort active move command and delete commands buffered in sequence
  /// No additional movements
  ABORT := 1,  
  /// 2: No reaction
  /// Error event is ignored by active move command
  NO_REACTION := 2
)USINT;
END_TYPE

// Library/Enumerations/Miscellaneous/LoadMeasurementSteps
{attribute 'qualified_only'}
// ------------------------------------------------------------------------- 
//  SRCI Robot Library                                                
// ------------------------------------------------------------------------- 
//                                                                           
//  Object:      LoadMeasurementSteps                                       
//  Author:      Thorsten Brach                                                
//  Date:        2024-06-01
//
//  Description:                                              
//   
//                                                                           
//  Copyright: 
//    (C) 2024 Thorsten Brach. All rights reserved                                                                                                                                            
//             Licensed under the LGPL-3.0 license.
//                                                                           
//  Disclaimer:                                                                           
//    This project is provided without any guarantee and can be used for   
//    private and commercial purposes. Any use is at the user’s 
//    own risk and responsibility.
//
// -------------------------------------------------------------------------
TYPE LoadMeasurementSteps :
(
  /// • 0: Reset (default)
  /// Delete all positions saved on the RC
  RESET := 0,  
  /// • 1: First position
  /// Save the first position for the load estimation with the required data
  FIRST_POSITION := 1,  
  /// • 2: Second position
  /// Save the second position for the load estimation with the required data
  SECOND_POSITION := 2,  
  /// • 3: Third position
  /// Save the third position for the load estimation with the required data
  THIRD_POSITION := 3,  
  /// • 4: Fourth position
  /// Save the fourth position for the load estimation with the required data
  FOURTH_POSITION := 4,  
  /// • 99: Load calculation
  /// Start the load calculation with the data saved in the four positions
  LOAD_CALCULATION := 99
)USINT;
END_TYPE

// Library/Enumerations/Miscellaneous/PathChoice
{attribute 'qualified_only'}
// ------------------------------------------------------------------------- 
//  SRCI Robot Library                                                
// ------------------------------------------------------------------------- 
//                                                                           
//  Object:      PathChoice                                       
//  Author:      Thorsten Brach                                                
//  Date:        2024-06-01
//
//  Description:                                              
//   
//                                                                           
//  Copyright: 
//    (C) 2024 Thorsten Brach. All rights reserved                                                                                                                                            
//             Licensed under the LGPL-3.0 license.
//                                                                           
//  Disclaimer:                                                                           
//    This project is provided without any guarantee and can be used for   
//    private and commercial purposes. Any use is at the user’s 
//    own risk and responsibility.
//
// -------------------------------------------------------------------------
TYPE PathChoice :
(
  /// Clockwise movement of the circular path
  CLOCKWISE := 0,
  /// Counterclockwise movement of the circular path
  COUNTERCLOCKWISE := 1
)BYTE;
END_TYPE

// Library/Enumerations/Miscellaneous/ReferenceElement
{attribute 'qualified_only'}
// ------------------------------------------------------------------------- 
//  SRCI Robot Library                                                
// ------------------------------------------------------------------------- 
//                                                                           
//  Object:      ReferenceElement                                       
//  Author:      Thorsten Brach                                                
//  Date:        2024-06-01
//
//  Description:                                              
//   
//                                                                           
//  Copyright: 
//    (C) 2024 Thorsten Brach. All rights reserved                                                                                                                                            
//             Licensed under the LGPL-3.0 license.
//                                                                           
//  Disclaimer:                                                                           
//    This project is provided without any guarantee and can be used for   
//    private and commercial purposes. Any use is at the user’s 
//    own risk and responsibility.
//
// -------------------------------------------------------------------------
TYPE ReferenceElement :
(
  /// 0 (default): Not used
  NOT_USED := 0,  
  /// 1: X-Axis
  X_AXIS := 1,
  /// 2: Y-Axis
  Y_AXIS := 2,
  /// 3: Z-Axis
  Z_AXIS := 3,
  /// 4: XY-Plane
  XY_PLANE := 4,
  /// 5: XZ-Plane
  XZ_PLANE := 5,
  /// 6: YZ-Plane
  YZ_PLANE := 6
)USINT;
END_TYPE

// Library/Enumerations/Miscellaneous/Severity
{attribute 'qualified_only'}
// ------------------------------------------------------------------------- 
//  SRCI Robot Library                                                
// ------------------------------------------------------------------------- 
//                                                                           
//  Object:      Severity                                       
//  Author:      Thorsten Brach                                                
//  Date:        2024-06-01
//
//  Description:                                              
//   
//                                                                           
//  Copyright: 
//    (C) 2024 Thorsten Brach. All rights reserved                                                                                                                                            
//             Licensed under the LGPL-3.0 license.
//                                                                           
//  Disclaimer:                                                                           
//    This project is provided without any guarantee and can be used for   
//    private and commercial purposes. Any use is at the user’s 
//    own risk and responsibility.
//
// -------------------------------------------------------------------------
TYPE Severity : 
(
  /// No events will be logged
  DEACTIVATE  := 0,
  /// Debug message
  /// • No user action required
  DEBUG := 4, 
  /// Informative message
  /// • No user action required
  INFO := 5,
  /// Warning message
  /// • User action will be required at some point
  WARNING := 20,
  /// Error message
  /// • User action required immediately
  ERROR := 28,
  ///  Fatal error message
  /// • User action required immediately
  /// • Reinitialization OF RI required
  FATAL_ERROR := 29
)SINT;
END_TYPE

// Library/Enumerations/Miscellaneous/SyncDirection
{attribute 'qualified_only'}
// ------------------------------------------------------------------------- 
//  SRCI Robot Library                                                
// ------------------------------------------------------------------------- 
//                                                                           
//  Object:      SyncDirection                                       
//  Author:      Thorsten Brach                                                
//  Date:        2024-06-01
//
//  Description:                                              
//   
//                                                                           
//  Copyright: 
//    (C) 2024 Thorsten Brach. All rights reserved                                                                                                                                            
//             Licensed under the LGPL-3.0 license.
//                                                                           
//  Disclaimer:                                                                           
//    This project is provided without any guarantee and can be used for   
//    private and commercial purposes. Any use is at the user’s 
//    own risk and responsibility.
//
// -------------------------------------------------------------------------
TYPE SyncDirection :
(
  /// No synchronization will be executed
  NO_SYNC := 0,
  /// Server data will be overwritten immediately by client data
  PLC_TO_ROB := 1,
  /// Client data will be overwritten immediately by server data
  ROB_TO_PLC := 2,
  /// Server or client data will be overwritten immediately by changed data
  AUTOMATIC := 3
);
END_TYPE

// Library/Enumerations/Miscellaneous/SyncReaction
{attribute 'qualified_only'}
// ------------------------------------------------------------------------- 
//  SRCI Robot Library                                                
// ------------------------------------------------------------------------- 
//                                                                           
//  Object:      SyncReaction                                       
//  Author:      Thorsten Brach                                                
//  Date:        2024-06-01
//
//  Description:                                              
//   
//                                                                           
//  Copyright: 
//    (C) 2024 Thorsten Brach. All rights reserved                                                                                                                                            
//             Licensed under the LGPL-3.0 license.
//                                                                           
//  Disclaimer:                                                                           
//    This project is provided without any guarantee and can be used for   
//    private and commercial purposes. Any use is at the user’s 
//    own risk and responsibility.
//
// -------------------------------------------------------------------------
TYPE SyncReaction :
(
  /// • System behavior unaffected
  NO_REACTION := 0,
  /// • No automatic disable
  /// • Reaction will only apply when RA is disabled
  /// • RA can only be enabled if client and server are synchronized
  REACTION_TYPE_1 := 1,  
  /// • No automatic disable
  /// • RA can only be enabled if client and server are synchronized
  /// • RA sequence state will change to interrupted when no command is buffered in the active sequence
  /// • Continuation is only possible if client and server are synchronized
  REACTION_TYPE_2 := 2,  
  /// • No automatic disable
  /// • RA can only be enabled if client and server are synchronized
  /// • RA sequence state will change to interrupted
  /// • Continuation is only possible if client and server are synchronized
  REACTION_TYPE_3 := 3
)USINT;
END_TYPE

// Library/Enumerations/Miscellaneous/TriggerCondition
{attribute 'qualified_only'}
// ------------------------------------------------------------------------- 
//  SRCI Robot Library                                                
// ------------------------------------------------------------------------- 
//                                                                           
//  Object:      TriggerCondition                                       
//  Author:      Thorsten Brach                                                
//  Date:        2024-06-01
//
//  Description:                                              
//   
//                                                                           
//  Copyright: 
//    (C) 2024 Thorsten Brach. All rights reserved                                                                                                                                            
//             Licensed under the LGPL-3.0 license.
//                                                                           
//  Disclaimer:                                                                           
//    This project is provided without any guarantee and can be used for   
//    private and commercial purposes. Any use is at the user’s 
//    own risk and responsibility.
//
// -------------------------------------------------------------------------
TYPE TriggerCondition :
(
  /// 5: Time in ms  - point reference is target position
  TARGET_POSITION_TIME_MS := -5,
  /// 4: TCP velocity in mm/s - point reference is target position
  TARGET_POSITION_TCP_VELOCITY_ABSOLUTE := -4,
  /// 3: TCP velocity in % of reference velocity - point reference is target position
  TARGET_POSITION_TCP_VELOCITY_PERCENT := -3,
  /// 2: Distance in mm of trajectory - point reference is target position
  TARGET_POSITION_DISTANCE_ABSOLUTE := -2,
  /// 1: Distance in % of trajectory - point reference is target position
  TARGET_POSITION_DISTANCE_PERCENT := -1,
  /// 0: Undfined 
  UNDEFINED := 0,
  /// 1: Distance in % of trajectory - point reference is start position
  START_POSITION_DISTANCE_PERCENT := 1,
  /// 2: Distance in mm of trajectory - point reference is start position
  START_POSITION_DISTANCE_ABSOLUTE := 2,
  /// 3: TCP velocity in % of reference velocity - point reference is start position
  START_POSITION_TCP_VELOCITY_PERCENT := 3,
  /// 4: TCP velocity in mm/s - point reference is start position
  START_POSITION_TCP_VELOCIT_ABSOLUTE := 4,
  /// 5: Time in ms - point reference is start position
  START_POSITION_TIME_MS := 5
)SINT;
END_TYPE

// Library/Enumerations/Mode/AbortingMode
{attribute 'qualified_only'}
// ------------------------------------------------------------------------- 
//  SRCI Robot Library                                                
// ------------------------------------------------------------------------- 
//                                                                           
//  Object:      AbortingMode                                       
//  Author:      Thorsten Brach                                                
//  Date:        2024-06-01
//
//  Description:                                              
//   
//                                                                           
//  Copyright: 
//    (C) 2024 Thorsten Brach. All rights reserved                                                                                                                                            
//             Licensed under the LGPL-3.0 license.
//                                                                           
//  Disclaimer:                                                                           
//    This project is provided without any guarantee and can be used for   
//    private and commercial purposes. Any use is at the user’s 
//    own risk and responsibility.
//
// -------------------------------------------------------------------------
TYPE AbortingMode :
(
  /// The current movement command as well as all stored movements are executed as programmed. 
  /// The new motion command is queued in the motion buffer.
  BUFFER := 0,
  /// The current movement command is aborted. All buffered motion movements are discarded. 
  /// The new target position is approached, depending on the motion command.
  ABORT  := 1
)SINT;
END_TYPE

// Library/Enumerations/Mode/BlendingMode
{attribute 'qualified_only'}
// ------------------------------------------------------------------------- 
//  SRCI Robot Library                                                
// ------------------------------------------------------------------------- 
//                                                                           
//  Object:      BlendingMode                                       
//  Author:      Thorsten Brach                                                
//  Date:        2024-06-01
//
//  Description:                                              
//   
//                                                                           
//  Copyright: 
//    (C) 2024 Thorsten Brach. All rights reserved                                                                                                                                            
//             Licensed under the LGPL-3.0 license.
//                                                                           
//  Disclaimer:                                                                           
//    This project is provided without any guarantee and can be used for   
//    private and commercial purposes. Any use is at the user’s 
//    own risk and responsibility.
//
// -------------------------------------------------------------------------
TYPE BlendingMode :
(
  /// Appended, buffered, no blending
  EXACT_STOP := 0,
  /// Start blending when the defined velocity is reached
  DEFINED_VELOCITY := 2,
  /// Define blending sphere with radius
  CORNER_DISTANCE := 3,
  /// Define blending with deviation
  MAX_CORNER_DEVIATION := 4,
  /// Define blending sphere with 2 radiuses
  CORNER_DISTANCE_2R := 10,
  /// Define blending with percentage of overlapping of deceleration and acceleration ramp
  RAMP_OVERLAP := 11,
  /// Define blending sphere with starting radius
  CORNER_DISTANCE_1R := 12
)USINT;
END_TYPE

// Library/Enumerations/Mode/CircMode
{attribute 'qualified_only'}
// ------------------------------------------------------------------------- 
//  SRCI Robot Library                                                
// ------------------------------------------------------------------------- 
//                                                                           
//  Object:      CircMode                                       
//  Author:      Thorsten Brach                                                
//  Date:        2024-06-01
//
//  Description:                                              
//   
//                                                                           
//  Copyright: 
//    (C) 2024 Thorsten Brach. All rights reserved                                                                                                                                            
//             Licensed under the LGPL-3.0 license.
//                                                                           
//  Disclaimer:                                                                           
//    This project is provided without any guarantee and can be used for   
//    private and commercial purposes. Any use is at the user’s 
//    own risk and responsibility.
//
// -------------------------------------------------------------------------
TYPE CircMode :
(
  /// "AuxPoint" defines a point on the circle crossed on the path from the starting to the end point.
  BORDER := 0,
  /// "AuxPoint" defines the center point of the circle.
  CENTER := 1,
  /// "AuxPoint" defines the center point of the circle, "Angle" defines the end position of the circular motion, and "CircPlane" defines the circle’s plane.
  CENTER_WITH_ANGLE := 2,
  /// "AuxPoint" defines a vector which length is the radius of the circle. The plane of the circle is defined by the rule of right thumb while the "AuxPoint" defines the spearhead point of the perpendicular.
  RADIUS := 3
)SINT;
END_TYPE

// Library/Enumerations/Mode/CollisionReactionMode
{attribute 'qualified_only'}
// ------------------------------------------------------------------------- 
//  SRCI Robot Library                                                
// ------------------------------------------------------------------------- 
//                                                                           
//  Object:      CollisionReactionMode                                       
//  Author:      Thorsten Brach                                                
//  Date:        2024-06-01
//
//  Description:                                              
//   
//                                                                           
//  Copyright: 
//    (C) 2024 Thorsten Brach. All rights reserved                                                                                                                                            
//             Licensed under the LGPL-3.0 license.
//                                                                           
//  Disclaimer:                                                                           
//    This project is provided without any guarantee and can be used for   
//    private and commercial purposes. Any use is at the user’s 
//    own risk and responsibility.
//
// -------------------------------------------------------------------------
TYPE CollisionReactionMode :
(
  /// Standing still
  STANDING_STILL := 0,
  /// Reversed movement
  REVERSED_MOVEMENT := 1
)USINT;
END_TYPE

// Library/Enumerations/Mode/ConnectionMode
{attribute 'qualified_only'}
// ------------------------------------------------------------------------- 
//  SRCI Robot Library                                                
// ------------------------------------------------------------------------- 
//                                                                           
//  Object:      ConnectionMode                                       
//  Author:      Thorsten Brach                                                
//  Date:        2024-06-01
//
//  Description:                                              
//   
//                                                                           
//  Copyright: 
//    (C) 2024 Thorsten Brach. All rights reserved                                                                                                                                            
//             Licensed under the LGPL-3.0 license.
//                                                                           
//  Disclaimer:                                                                           
//    This project is provided without any guarantee and can be used for   
//    private and commercial purposes. Any use is at the user’s 
//    own risk and responsibility.
//
// -------------------------------------------------------------------------
TYPE ConnectionMode :
(
  /// Encoder is connected to RC
  RC_CONNECTED := 0,
  /// Encoder is connected to PLC
  PLC_CONNECTED := 1
)SINT;
END_TYPE

// Library/Enumerations/Mode/DefinitionMode
{attribute 'qualified_only'}
// ------------------------------------------------------------------------- 
//  SRCI Robot Library                                                
// ------------------------------------------------------------------------- 
//                                                                           
//  Object:      DefinitionMode                                       
//  Author:      Thorsten Brach                                                
//  Date:        2024-06-01
//
//  Description:                                              
//   
//                                                                           
//  Copyright: 
//    (C) 2024 Thorsten Brach. All rights reserved                                                                                                                                            
//             Licensed under the LGPL-3.0 license.
//                                                                           
//  Disclaimer:                                                                           
//    This project is provided without any guarantee and can be used for   
//    private and commercial purposes. Any use is at the user’s 
//    own risk and responsibility.
//
// -------------------------------------------------------------------------
TYPE DefinitionMode :
(
  /// ZeroPoint describes center point of body 
  Center := 1,
  /// ZeroPoint describes point on face of body. Parameter values for X2, Y2, Z2 will be ignored  
  Face := 2 
)USINT;
END_TYPE

// Library/Enumerations/Mode/DetectionMode
{attribute 'qualified_only'}
// ------------------------------------------------------------------------- 
//  SRCI Robot Library                                                
// ------------------------------------------------------------------------- 
//                                                                           
//  Object:      DetectionMode                                       
//  Author:      Thorsten Brach                                                
//  Date:        2024-06-01
//
//  Description:                                              
//   
//                                                                           
//  Copyright: 
//    (C) 2024 Thorsten Brach. All rights reserved                                                                                                                                            
//             Licensed under the LGPL-3.0 license.
//                                                                           
//  Disclaimer:                                                                           
//    This project is provided without any guarantee and can be used for   
//    private and commercial purposes. Any use is at the user’s 
//    own risk and responsibility.
//
// -------------------------------------------------------------------------
TYPE DetectionMode :
(
  /// Torque (default)
  TORQUE := 0,
  /// Force
  FORCE := 1,
  /// Electrical current
  ELECTRICAL_CURRENT := 2,
  /// Following Error
  FOLLOWING_ERROR := 3
)USINT;
END_TYPE

// Library/Enumerations/Mode/ErrorTriggerMode
{attribute 'qualified_only'}
// ------------------------------------------------------------------------- 
//  SRCI Robot Library                                                
// ------------------------------------------------------------------------- 
//                                                                           
//  Object:      ErrorTriggerMode                                       
//  Author:      Thorsten Brach                                                
//  Date:        2024-06-01
//
//  Description:                                              
//   
//                                                                           
//  Copyright: 
//    (C) 2024 Thorsten Brach. All rights reserved                                                                                                                                            
//             Licensed under the LGPL-3.0 license.
//                                                                           
//  Disclaimer:                                                                           
//    This project is provided without any guarantee and can be used for   
//    private and commercial purposes. Any use is at the user’s 
//    own risk and responsibility.
//
// -------------------------------------------------------------------------
TYPE ErrorTriggerMode :
(
  /// Any command (default)
  ANY_COMMAND := 0,
  /// General commands
  GENERAL_COMMANDS := 1,
  /// Administrative commands
  ADMINISTRATIVE_COMMANDS := 2,
  /// Move commands
  MOVE_COMMANDS := 3,
  /// Periphery commands
  PERIPHERY_COMMANDS := 4,
  /// Extended commands
  EXTENDED_COMMANDS := 5,
  /// Specific command or RI message
  SPECIFIC_COMMAND_OR_RI_MESSAGE := 6,
  /// Specific RC or RA message code
  SPECIFIC_RC_OR_RA_MESSAGE_CODE := 7,
  /// Any RI message code
  ANY_RI_MESSAGE_CODE := 8,
  /// Any RC or RA message code
  ANY_RC_OR_RA_MESSAGE_CODE := 9
)SINT;
END_TYPE

// Library/Enumerations/Mode/ExecutionMode
{attribute 'qualified_only'}
// ------------------------------------------------------------------------- 
//  SRCI Robot Library                                                
// ------------------------------------------------------------------------- 
//                                                                           
//  Object:      ExecutionMode                                       
//  Author:      Thorsten Brach                                                
//  Date:        2024-06-01
//
//  Description:                                              
//   
//                                                                           
//  Copyright: 
//    (C) 2024 Thorsten Brach. All rights reserved                                                                                                                                            
//             Licensed under the LGPL-3.0 license.
//                                                                           
//  Disclaimer:                                                                           
//    This project is provided without any guarantee and can be used for   
//    private and commercial purposes. Any use is at the user’s 
//    own risk and responsibility.
//
// -------------------------------------------------------------------------
TYPE ExecutionMode :
(
  /// Command is buffered in sequence buffer and executed once
  SEQUENCE_PRIMARY := 0,
  /// Command is buffered in sequence buffer, aborts and empties previous commands in sequence buffer, and is executed once
  SEQUENCE_ABORT_OTHERS_PRIMARY := 1,
  /// Command is buffered in parallel buffer and executed once. The execution may also be Trigger based.
  PARALLEL := 2,
  /// Command is buffered in parallel buffer and executed repeatedly until deliberate deactivation by user. The de- and activation may also be Trigger based.
  CONTINUOUS := 3,
  /// Command is buffered and executed once when triggered. The CMD remains in the buffer until removed by the user.
  TRIGGER_MULTIPLE := 5,
  /// Command is buffered in sequence buffer and executed once (Secondary)
  SEQUENCE_SECONDARY := 7,
  /// Command is buffered in sequence buffer, aborts and empties previous commands in sequence buffer and is executed once (Secondary)
  SEQUENCE_ABORT_OTHERS_SECONDARY := 8,
  /// CMD execution is stopped and/or CMD is removed from the buffer.
  STOP_PARALLEL_CONTINUOUS_TRIGGER := 9
)USINT;
END_TYPE

// Library/Enumerations/Mode/FrameCalculationMode
{attribute 'qualified_only'}
// ------------------------------------------------------------------------- 
//  SRCI Robot Library                                                
// ------------------------------------------------------------------------- 
//                                                                           
//  Object:      FrameCalculationMode                                       
//  Author:      Thorsten Brach                                                
//  Date:        2024-06-01
//
//  Description:                                              
//   
//                                                                           
//  Copyright: 
//    (C) 2024 Thorsten Brach. All rights reserved                                                                                                                                            
//             Licensed under the LGPL-3.0 license.
//                                                                           
//  Disclaimer:                                                                           
//    This project is provided without any guarantee and can be used for   
//    private and commercial purposes. Any use is at the user’s 
//    own risk and responsibility.
//
// -------------------------------------------------------------------------
TYPE FrameCalculationMode :
(
  /// 0: Three-Point-method (default)
  THREE_POINT_METHOD := 0,  
  /// 1: Four-Point-method
  FOUR_POINT_METHOD := 1,  
  /// 2: One-Point-method
  ONE_POINT_METHOD := 2
)SINT;
END_TYPE

// Library/Enumerations/Mode/FunctionMode
{attribute 'qualified_only'}
// ------------------------------------------------------------------------- 
//  SRCI Robot Library                                                
// ------------------------------------------------------------------------- 
//                                                                           
//  Object:      FunctionMode                                       
//  Author:      Thorsten Brach                                                
//  Date:        2024-06-01
//
//  Description:                                              
//   
//                                                                           
//  Copyright: 
//    (C) 2024 Thorsten Brach. All rights reserved                                                                                                                                            
//             Licensed under the LGPL-3.0 license.
//                                                                           
//  Disclaimer:                                                                           
//    This project is provided without any guarantee and can be used for   
//    private and commercial purposes. Any use is at the user’s 
//    own risk and responsibility.
//
// -------------------------------------------------------------------------
TYPE FunctionMode :
(
  enum_member := 0
);
END_TYPE

// Library/Enumerations/Mode/InterpolationMode
{attribute 'qualified_only'}
// ------------------------------------------------------------------------- 
//  SRCI Robot Library                                                
// ------------------------------------------------------------------------- 
//                                                                           
//  Object:      InterpolationMode                                       
//  Author:      Thorsten Brach                                                
//  Date:        2024-06-01
//
//  Description:                                              
//   
//                                                                           
//  Copyright: 
//    (C) 2024 Thorsten Brach. All rights reserved                                                                                                                                            
//             Licensed under the LGPL-3.0 license.
//                                                                           
//  Disclaimer:                                                                           
//    This project is provided without any guarantee and can be used for   
//    private and commercial purposes. Any use is at the user’s 
//    own risk and responsibility.
//
// -------------------------------------------------------------------------
TYPE InterpolationMode :
(
  /// Linear interpolation
  Linear_interpolation := 0,
  /// Direct interpolation (PTP)
  Direct_interpolation := 1
)USINT;
END_TYPE

// Library/Enumerations/Mode/JogMode
{attribute 'qualified_only'}
// ------------------------------------------------------------------------- 
//  SRCI Robot Library                                                
// ------------------------------------------------------------------------- 
//                                                                           
//  Object:      JogMode                                       
//  Author:      Thorsten Brach                                                
//  Date:        2024-06-01
//
//  Description:                                              
//   
//                                                                           
//  Copyright: 
//    (C) 2024 Thorsten Brach. All rights reserved                                                                                                                                            
//             Licensed under the LGPL-3.0 license.
//                                                                           
//  Disclaimer:                                                                           
//    This project is provided without any guarantee and can be used for   
//    private and commercial purposes. Any use is at the user’s 
//    own risk and responsibility.
//
// -------------------------------------------------------------------------
TYPE JogMode :
(
  /// • Jog TCP manually in the given frame (WCS/UCS)
  /// • Movement on several coordinate axes simultaneously possible
  JOG_FRAME := 0,
  /// • Jog TCP manually in the given tool coordinate system
  /// • Movement on several coordinate axes simultaneously possible
  JOG_TOOL := 1,
  /// • Jog joints manually without referring to a given frame or tool
  /// • Movement of several axes simultaneously possible.
  JOG_AXES := 2
)USINT;
END_TYPE

// Library/Enumerations/Mode/LimitMode
{attribute 'qualified_only'}
// ------------------------------------------------------------------------- 
//  SRCI Robot Library                                                
// ------------------------------------------------------------------------- 
//                                                                           
//  Object:      LimitMode                                       
//  Author:      Thorsten Brach                                                
//  Date:        2024-06-01
//
//  Description:                                              
//   
//                                                                           
//  Copyright: 
//    (C) 2024 Thorsten Brach. All rights reserved                                                                                                                                            
//             Licensed under the LGPL-3.0 license.
//                                                                           
//  Disclaimer:                                                                           
//    This project is provided without any guarantee and can be used for   
//    private and commercial purposes. Any use is at the user’s 
//    own risk and responsibility.
//
// -------------------------------------------------------------------------
TYPE LimitMode :
(
  /// 0: No limit defined (default)
  /// The robot can be moved in the direction set with the input parameter "CompliantAxes" in a compliant manner by applying an external force on it.
  /// By reaching the mechanical or software limits, the robot stops.
  NO_LIMIT_DEFINED := 0,
  
  /// 1: Limit defined
  /// The robot can be moved along the defined vector in a compliant manner by applying an external force on it.
  /// By reaching the vector limit defined by the input parameter "VectorData", the robot stops.
  LIMIT_DEFINED := 1
)USINT;
END_TYPE

// Library/Enumerations/Mode/LoadMeasurementMode
{attribute 'qualified_only'}
// ------------------------------------------------------------------------- 
//  SRCI Robot Library                                                
// ------------------------------------------------------------------------- 
//                                                                           
//  Object:      LoadMeasurementMode                                       
//  Author:      Thorsten Brach                                                
//  Date:        2024-06-01
//
//  Description:                                              
//   
//                                                                           
//  Copyright: 
//    (C) 2024 Thorsten Brach. All rights reserved                                                                                                                                            
//             Licensed under the LGPL-3.0 license.
//                                                                           
//  Disclaimer:                                                                           
//    This project is provided without any guarantee and can be used for   
//    private and commercial purposes. Any use is at the user’s 
//    own risk and responsibility.
//
// -------------------------------------------------------------------------
TYPE  LoadMeasurementMode :
(
  /// 0: One Position (default)
  /// Use one defined position and optional axes ranges
  ONE_POSITION := 0,  
  /// 1: Configuration Angle
  /// Use one defined position and optional axes ranges
  CONFIGURATION_ANGLE := 1,  
  /// 2: Area
  /// Use a defined area for the measurement
  AREA := 2,  
  /// 3: Two Positions
  /// Use defined positions for the measurement
  TWO_POSITIONS := 3
)USINT;
END_TYPE

// Library/Enumerations/Mode/LogonMode
{attribute 'qualified_only'}
// ------------------------------------------------------------------------- 
//  SRCI Robot Library                                                
// ------------------------------------------------------------------------- 
//                                                                           
//  Object:      LogonMode                                       
//  Author:      Thorsten Brach                                                
//  Date:        2024-06-01
//
//  Description:                                              
//   
//                                                                           
//  Copyright: 
//    (C) 2024 Thorsten Brach. All rights reserved                                                                                                                                            
//             Licensed under the LGPL-3.0 license.
//                                                                           
//  Disclaimer:                                                                           
//    This project is provided without any guarantee and can be used for   
//    private and commercial purposes. Any use is at the user’s 
//    own risk and responsibility.
//
// -------------------------------------------------------------------------
TYPE LogonMode :
(
  /// Password only (default)
  PASSWORD_ONLY := 0,
  /// Username and Password
  USERNAME_AND_PASSWORD := 1,
  /// Level ID and Password
  LEVEL_ID_AND_PASSWORD := 2
)SINT;
END_TYPE

// Library/Enumerations/Mode/MeasuringIoMode
{attribute 'qualified_only'}
// ------------------------------------------------------------------------- 
//  SRCI Robot Library                                                
// ------------------------------------------------------------------------- 
//                                                                           
//  Object:      MeasuringIoMode                                       
//  Author:      Thorsten Brach                                                
//  Date:        2024-06-01
//
//  Description:                                              
//   
//                                                                           
//  Copyright: 
//    (C) 2024 Thorsten Brach. All rights reserved                                                                                                                                            
//             Licensed under the LGPL-3.0 license.
//                                                                           
//  Disclaimer:                                                                           
//    This project is provided without any guarantee and can be used for   
//    private and commercial purposes. Any use is at the user’s 
//    own risk and responsibility.
//
// -------------------------------------------------------------------------
TYPE MeasuringIoMode :
(
  /// Measurement at next rising edge 
  /// • Output "MeasuredPosition_1" used
  MEASUREMENT_AT_NEXT_RISING_EDGE := 0,
  /// Measurement at next falling edge 
  /// • Output "MeasuredPosition_1" used
  MEASUREMENT_AT_NEXT_FALLING_EDGE := 1,
  /// Measurement at next edges, regardless of rising or falling edges.
  /// • First position stored in output "MeasuredPosition_1"
  /// • Second position stored in output "MeasuredPosition_2"
  MEASUREMENT_AT_NEXT_EDGE := 2,
  /// Measurement at two edges, beginning with the rising edge:
  /// • Rising edge = "MeasuredPosition_1 "
  /// • Falling edge = "MeasuredPosition_2 "
  MEASUREMENT_AT_TWO_EDGES_BEGIN_WITH_RISING := 3,
  /// Measurement at two edges, beginning with the falling edge:
  /// • Falling edge = " MeasuredPosition_1 "
  /// • Rising edge = "MeasuredPosition_2 "
  MEASUREMENT_AT_TWO_EDGES_BEGIN_WITH_FALLING := 4
)USINT;
END_TYPE

// Library/Enumerations/Mode/MeasuringUnitMode
{attribute 'qualified_only'}
// ------------------------------------------------------------------------- 
//  SRCI Robot Library                                                
// ------------------------------------------------------------------------- 
//                                                                           
//  Object:      MeasuringUnitMode                                       
//  Author:      Thorsten Brach                                                
//  Date:        2024-06-01
//
//  Description:                                              
//   
//                                                                           
//  Copyright: 
//    (C) 2024 Thorsten Brach. All rights reserved                                                                                                                                            
//             Licensed under the LGPL-3.0 license.
//                                                                           
//  Disclaimer:                                                                           
//    This project is provided without any guarantee and can be used for   
//    private and commercial purposes. Any use is at the user’s 
//    own risk and responsibility.
//
// -------------------------------------------------------------------------
TYPE MeasuringUnitMode :
(
  /// 0: VectorLength (default)
  ///    Defines the distance in millimeter between two points in cartesian space.
  VECTOR_LENGTH  := 0,
  /// 1: SegmentLength
  ///    Defines the distance in mm covered between the two points in cartesian space
  SEGMENT_LENGTH := 1,
  /// 2: Time
  ///    Defines the duration in milliseconds between the start and end point.
  TIME_DURATION  := 2
)USINT;
END_TYPE

// Library/Enumerations/Mode/OperationMode
{attribute 'qualified_only'}
// ------------------------------------------------------------------------- 
//  SRCI Robot Library                                                
// ------------------------------------------------------------------------- 
//                                                                           
//  Object:      OperationMode                                       
//  Author:      Thorsten Brach                                                
//  Date:        2024-06-01
//
//  Description:                                              
//   
//                                                                           
//  Copyright: 
//    (C) 2024 Thorsten Brach. All rights reserved                                                                                                                                            
//             Licensed under the LGPL-3.0 license.
//                                                                           
//  Disclaimer:                                                                           
//    This project is provided without any guarantee and can be used for   
//    private and commercial purposes. Any use is at the user’s 
//    own risk and responsibility.
//
// -------------------------------------------------------------------------
TYPE OperationMode :
(
 /// Test mode 1:
 /// • Maximum velocity of TCP is restricted to <250 mm/s
 /// • Robot can only be moved while enable switch is active
 /// • Designed for jogging, teaching program, verification
 /// • Safety door can be opened
 T1_LOCAL := 1,
 /// Test mode 2:
 /// • Maximum velocity of TCP not restricted (100%)
 /// • Robot can only be moved while enable switch is active
 /// • Designed for program verification (step mode)
 /// • Safety door can be opened
 T2_LOCAL := 2,
 /// Automatic mode:
 /// • Maximum velocity of TCP not restricted (100%)
 /// • Robot is executing user program automatically
 /// • Robot will stop if safety devices report error (e.g. safety door must be closed)
 AUTO := 3,
 /// External Automatic mode (PLC mode)
 /// • Robot is operated remotely only
 /// • Maximum velocity of TCP not restricted (100%)
 /// • Robot is executing user program automatically
 /// • Jogging possible
 /// • Robot will stop if safety devices report error (e.g. safety door must be closed)
 AUTO_EXT := 4,
 /// External Test mode 1 (PLC mode with T1 functionality)
 /// • Robot is operated remotely only
 /// • Maximum velocity of TCP is restricted to <250 mm/s
 /// • Robot can only be moved while enable switch is active
 /// • Designed for jogging, teaching, program verification
 /// • Safety door can be opened
 T1_EXT := 5,
 /// External Test mode 2:
 /// • Robot is operated remotely only
 /// • Maximum velocity of TCP not restricted (100%)
 /// • Robot can only be moved while enable switch is active
 /// • Designed for jogging, program verification (step mode)
 /// • Safety door can be opened
 T2_EXT := 6
)USINT;
END_TYPE

// Library/Enumerations/Mode/OrientationMode
{attribute 'qualified_only'}
// ------------------------------------------------------------------------- 
//  SRCI Robot Library                                                
// ------------------------------------------------------------------------- 
//                                                                           
//  Object:      OrientationMode                                       
//  Author:      Thorsten Brach                                                
//  Date:        2024-06-01
//
//  Description:                                              
//   
//                                                                           
//  Copyright: 
//    (C) 2024 Thorsten Brach. All rights reserved                                                                                                                                            
//             Licensed under the LGPL-3.0 license.
//                                                                           
//  Disclaimer:                                                                           
//    This project is provided without any guarantee and can be used for   
//    private and commercial purposes. Any use is at the user’s 
//    own risk and responsibility.
//
// -------------------------------------------------------------------------
TYPE OrientationMode :
(
    /// Change orientation continuously in a linear way
    LINEAR_INTERPOLATED := 1,
    /// Change orientation continuously in a joint interpolated way of wrist joints
    JOINT_INTERPOLATED := 2,
    /// No change of orientation during movement
    FIX := 3,
    /// No change of orientation in relation to trajectory
    PATH := 4
)SINT;
END_TYPE

// Library/Enumerations/Mode/OriMode
{attribute 'qualified_only'}
// ------------------------------------------------------------------------- 
//  SRCI Robot Library                                                
// ------------------------------------------------------------------------- 
//                                                                           
//  Object:      OriMode                                       
//  Author:      Thorsten Brach                                                
//  Date:        2024-06-01
//
//  Description:                                              
//   
//                                                                           
//  Copyright: 
//    (C) 2024 Thorsten Brach. All rights reserved                                                                                                                                            
//             Licensed under the LGPL-3.0 license.
//                                                                           
//  Disclaimer:                                                                           
//    This project is provided without any guarantee and can be used for   
//    private and commercial purposes. Any use is at the user’s 
//    own risk and responsibility.
//
// -------------------------------------------------------------------------
TYPE OriMode :
(
  /// Change orientation continuously in a linear way
  LINEAR_INTERPOLATED := 1,
  /// Change orientation continuously in a joint interpolated way.
  JOINT_INTERPOLATED  := 2,
  /// No change of orientation during movement
  FIX                 := 3,
  /// No change of orientation in relation to trajectory
  PATH                := 4
)USINT;
END_TYPE

